{attribute addProperty BoxType "KL2531-0001"}
{attribute addProperty Id "Channel_1Channel_55398A3800"}
{attribute addProperty CRC "1172248193"}
{attribute addProperty SizeInBites "0"}
{attribute addProperty SizeInBytes "0"}
TYPE KL_45DF1681 :
STRUCT
	{attribute addProperty Name "Channel_1"}
	Channel_1 : Channel_55398A38;
END_STRUCT
END_TYPE

(* stored: Version 1.2.0.0, ProductVersion 3.1.4024.9
   DUT KL_45DF1681: Id {aaaf5b3c-3712-4d9c-be09-d6a94afbf63f} *)
